FUNCTION_BLOCK TRingCounter_UDINT
VAR
    Count : UDINT;
    _StartValue : UDINT;
    _EndValue : UDINT;
END_VAR

PROPERTY EndValue : UDINT
GET
EndValue := _EndValue;
END_GET
SET
_EndValue := EndValue;
END_SET
END_PROPERTY

METHOD FB_init : BOOL
VAR_INPUT
	bInitRetains : BOOL; // if TRUE, the retain variables are initialized (warm start / cold start)
	bInCopyCode : BOOL;  // if TRUE, the instance afterwards gets moved into the copy code (online change)

    StartValue : UDINT;
    EndValue : UDINT;
END_VAR
THIS^._StartValue := StartValue;
THIS^._EndValue := EndValue;
Reset();
END_METHOD

METHOD Inc
VAR_INPUT
END_VAR
Count := Count + 1;
IF Count > EndValue THEN
    Reset();
END_IF
END_METHOD

PROPERTY NextValue : UDINT
GET
IF Count = EndValue THEN
    NextValue := StartValue;
ELSE
    NextValue := Count + 1;
END_IF
END_GET
END_PROPERTY

METHOD Reset
VAR_INPUT
END_VAR
Count := StartValue;
END_METHOD

PROPERTY StartValue : UDINT
GET
StartValue := _StartValue;
END_GET
SET
_StartValue := StartValue;
END_SET
END_PROPERTY

PROPERTY Value : UDINT
GET
Value := Count;
END_GET
SET
Count := Value;
END_SET
END_PROPERTY

END_FUNCTION_BLOCK

(* stored: Version 1.1.0.1, ProductVersion 3.1.4024.3
   POU TRingCounter_UDINT: Id {4ca36dc5-5a44-0804-090d-0b63699fa46a}, SpecialFunc None
   Folder Methods: Id {56069032-0dd3-0f39-1732-cdf7de423bba}
   Folder Properties: Id {9defc9bb-c28f-0581-2e66-adac7c420a6e}
   Property EndValue: Id {9de22e34-012e-03b6-2b7c-d791981813fb}
   Get Get: Id {398f041e-1bb3-0516-2b49-fbad9651267f}
   Set Set: Id {988ece23-c5a5-0c24-2404-fae2da3fcc4b}
   Method FB_init: Id {a10de747-59ed-016d-09c2-801f322b0673}
   Method Inc: Id {e823e340-c4e5-0d04-3275-6ab22e99868e}
   Property NextValue: Id {480d66a8-6e2e-0455-0f0f-6f8937bc263d}
   Get Get: Id {a02dd428-6145-0eb1-15f0-cd3a6b042ce2}
   Method Reset: Id {5e5cf99f-b4cb-0f19-1f7d-0862ee9df79b}
   Property StartValue: Id {4bc46c8f-96d3-01d9-1e94-6754a7523c86}
   Get Get: Id {0d928486-c844-0a53-3ce7-c72b1c7689c7}
   Set Set: Id {b4960e87-45c0-0085-0e42-c9e0895d22f3}
   Property Value: Id {6a69f0cd-3137-0cc8-08b6-539c3db66e18}
   Get Get: Id {83452381-24c0-02bf-159d-2f0b94907bf5}
   Set Set: Id {00ca97aa-6afa-0a2d-2fb0-72dee1512352} *)
